TYPE ST_ElementMemberList :
(**************************************************************************************
 * 	Application		:	BoxControl Framework
 *	Revision		:	$Revision: 404529 $
 *	Revision date	:	$Date: 2018-04-23 08:21:38 +0200 (Mo., 23 Apr 2018) $
 *	Last changed by	:	$Author: b7bolm $
 *	URL				:	$URL: http://almscdc.swisslog.com/repo/SWPD/Development/BoxControlFramework/20_Release/trunk/01_Software/BCF/BCF/JumpStart/20_Product/10_App/13_Elements/10_Lib/10_Conv/01_DUTs/ST_ElementMemberList.TcDUT $
 *
 *	Purpose			:	List of members which are linked to a element
 *
 * ------------------------------------------------------------------------------------
 *	Copyright Swisslog [IP AG], Switzerland. All rights reserved.
 * 
 * ------------------------------------------------------------------------------------
 *	
 * 	Revision History: 
 *
 * 	VERSION			DATE			INITIALS			DESCRIPTION
 *	0.1				01.01.2001		swl					Example
 *
 **************************************************************************************)
STRUCT
	FunctionList		: ARRAY [1 .. NUMBER_OF_FUNCTIONS_PER_ELEMENT] OF ST_FunctionEntry; // Registred function to this element
	ElementList			: ST_ElementMasterSlave; // Element slave
END_STRUCT
END_TYPE

(* stored: Version 1.1.0.1, ProductVersion 3.1.4022.12
   DUT ST_ElementMemberList: Id {7c1264c8-ae00-4602-9aab-596efbb03014} *)
